(* IEC 61131-3 sources: RPA_SEM_TRYSKANI/, 5 files *)

(* ---- piskovani_new_pokus.st ---- *)
TYPE
  SuperStatesEnum : (ST_INICIALIZACE, ST_RESET_POSITION_OF_MOTORS, ST_WAIT_FOR_COMMAND, ST_MODE_SELECTION, ST_MANUAL_MODE, ST_AUTOMATIC_MODE, ST_CHECK_POSITION_OF_MOTORS, ST_STOP, ST_EMERGENCY_STOP) := ST_INICIALIZACE;
END_TYPE

PROGRAM SuperStavy
  VAR
    I_Start AT %IX0.6 : BOOL := 1;
    I_PowerOn AT %IX1.1 : BOOL := 1;
    I_StopBtn AT %IX1.2 : BOOL;
    I_StopResBtn AT %IX1.3 : BOOL;
    I_EmStopBtn AT %IX1.4 : BOOL;
    I_EmStopResBtn AT %IX1.5 : BOOL;
    I_ManualSelector AT %IX1.6 : BOOL;
    I_AutomaticSelector AT %IX1.7 : BOOL := 1;
  END_VAR
  VAR
    SuperStates : SuperStatesEnum := ST_INICIALIZACE;
  END_VAR
  VAR
    I_A0 AT %IX0.0 : BOOL;
    I_A1 AT %IX0.1 : BOOL;
    I_B0 AT %IX0.2 : BOOL;
    I_B1 AT %IX0.3 : BOOL;
    I_C0 AT %IX0.4 : BOOL;
    I_C1 AT %IX0.5 : BOOL;
  END_VAR
  VAR
    I_Qt : BOOL;
  END_VAR
  VAR
    Q_A AT %QX0.4 : BOOL;
    Q_B AT %QX0.5 : BOOL;
    Q_C AT %QX0.6 : BOOL;
  END_VAR
  VAR
    Q_PositionOk : BOOL;
    Q_PositionNotOk : BOOL;
    Q_It : BOOL;
    InputArr : ARRAY [0..7] OF BYTE;
    InputWord : INT;
    TRANS_MATX : ARRAY [0..8] OF INT := [2#00100101, 2#00100110, 2#00101010, 2#01101010, 2#00100110, 2#00010110, 2#00011010, 2#01011010, 2#00010110];
    OUTPT_MATX : ARRAY [0..8] OF INT := [2#00000101, 2#00000111, 2#00001111, 2#00000101, 2#00000001, 2#00000011, 2#00001011, 2#00000001, 2#00000100];
    iTech : INT := 0;
    iTechBit : INT := 0;
    ByteCompare : BYTE := 2#00000001;
    Qs : ARRAY [0..7] OF BOOL;
    TechnologicalSequenceState : INT := 0;
    SuperSequenceState : INT := 1;
    TON_0 : TON;
    BlastingTime : TIME := t#5s;
  END_VAR

  (*IF (I_EMSTOPBTN = true) THEN

      SuperStates := ST_EMERGENCY_STOP;

  END_IF;*)

  IF (I_Start = true) THEN

      SuperStates := ST_INICIALIZACE;

  ELSE
      SuperStates := ST_STOP;

  END_IF;

  CASE SuperStates OF

    ST_INICIALIZACE:
      (*SuperSequenceState := 1;
      IF (I_Start = true) THEN (*Uprava 06.05.2021*)

        (*SuperStates := ST_RESET_POSITION_OF_MOTORS;

      END_IF;*)

      SuperStates := ST_RESET_POSITION_OF_MOTORS;

    ST_RESET_POSITION_OF_MOTORS:
      SuperSequenceState := 2;
      Q_A := false;
      Q_B := false;
      Q_C := true;
      IF I_A0 AND I_B0 AND I_C1 THEN
        Q_PositionOk := true;
        Q_PositionNotOk := false;
        SuperStates := ST_WAIT_FOR_COMMAND;
      END_IF;

    ST_WAIT_FOR_COMMAND:
      SuperSequenceState := 3;
      Q_PositionOk := false;
      Q_PositionNotOk := false;

      SuperStates := ST_MODE_SELECTION;

    ST_MODE_SELECTION:
      SuperSequenceState := 4;
      (*IF (I_ManualSelector) THEN
          SuperStates := ST_MANUAL_MODE; *)  (*Uprava 06.05.2021*)
      (*ELSIF (I_AutomaticSelector) THEN *)
      IF (I_Start = true) THEN
          SuperStates := ST_AUTOMATIC_MODE;
      ELSIF (I_ManualSelector = true) AND (I_Start = true) THEN
          SuperStates := ST_MANUAL_MODE;
      END_IF;

      (*END_IF;*)    (*Uprava 06.05.2021*)
      (*TODO// Comeback from this state to STOP*)

    ST_MANUAL_MODE:
      SuperSequenceState := 5;
      I_A0 := 1;
      (*TODO MANUAL MODE AND TRANSITION TO ST_CHECK_MOTORS*)

    ST_AUTOMATIC_MODE:
      SuperSequenceState := 6;

      (*  Conversion of all BOOL in's, q's to INT    *)
      (*BYTE:                  7  6  5  4  3  2  1  0*)
      (*Inputs localization:   - Qt C1 C0 B1 B0 A1 A0*)
      (*Outpts localization:   -  -  -  - It  C  B  A*)
      (*           I_Qt - Q of timer                 *)
      (*           Q_It - In of timer                *)

      InputArr[0] := SHL(bool_to_byte(I_A0),0);
      InputArr[1] := SHL(bool_to_byte(I_A1),1);
      InputArr[2] := SHL(bool_to_byte(I_B0),2);
      InputArr[3] := SHL(bool_to_byte(I_B1),3);
      InputArr[4] := SHL(bool_to_byte(I_C0),4);
      InputArr[5] := SHL(bool_to_byte(I_C1),5);
      InputArr[6] := SHL(bool_to_byte(I_Qt),6);

      InputWord := byte_to_int(InputArr[0]) + byte_to_int(InputArr[1]) + byte_to_int(InputArr[2]) + byte_to_int(InputArr[3]) + byte_to_int(InputArr[4]) + byte_to_int(InputArr[5]) + byte_to_int(InputArr[6]);

      (*   End of Conversion   *)

      IF (InputWord = TRANS_MATX[iTech]) THEN

        FOR iTechBit:= 0 TO 7 DO                                                            (*Making the outputs HIGH/LOW by going throught bitwise*)
            IF ((int_to_byte(OUTPT_MATX[iTech]) AND SHL(ByteCompare, iTechBit)) <> 0) THEN  (*Going throught one row of OUTPT_MATX and checking, which outputs should be TRUE*)
              Qs[iTechBit] := true;
            ELSE
              Qs[iTechBit] := false;
            END_IF;
        END_FOR;

        (*Mapping of outputs*)
        Q_A := Qs[0];
        Q_B := Qs[1];
        Q_C := Qs[2];
        Q_It := Qs[3];
        (*End of mapping of outputs*)

        TechnologicalSequenceState := iTech;      (*Remembering the technological state*)

        iTech := iTech + 1;                       (*Going to the next state*)

      END_IF;

      (*Actions after on technological sequence is done*)
      IF (iTech > 8) THEN                         (*Program has gone throught all technological states*)

        iTech := 0;                               (*Reset sequence*)
      END_IF;

     (*ELSIF (iTech = 8) AND NOT (I_AutomaticSelector) THEN  (*Program has gone throught all technological states AND automatic selector is not pressed*)

      (*  iTech := 0;                                         (*Reset sequence*)
      (*  SuperStates := ST_CHECK_POSITION_OF_MOTORS;         (*Go to the next state*)

      (*ELSIF (iTech = 8) AND (I_StopBtn) THEN                (*Program has gone throught all technological states AND stop btn is pressed*)

       (* SuperStates := ST_STOP;                               (*Go to stop state*)

     (* END_IF;*)

    ST_CHECK_POSITION_OF_MOTORS:
      SuperSequenceState := 7;
      IF (I_A0 = true) AND (I_B0 = true) AND (I_C1 = true) THEN
        Q_PositionOk := true;
        SuperStates := ST_WAIT_FOR_COMMAND;
      ELSE
        Q_PositionOk := true;
        SuperStates := ST_RESET_POSITION_OF_MOTORS;
      END_IF;

    ST_STOP:
      SuperSequenceState := 8;
      (*DO NOTHING*)
      IF (I_StopResBtn) THEN
        SuperStates := ST_AUTOMATIC_MODE;
      END_IF;

    ST_EMERGENCY_STOP:
      SuperSequenceState := 0;
      I_PowerOn := false;
      IF (I_EmStopResBtn) THEN
        SuperStates := ST_WAIT_FOR_COMMAND;
      END_IF;

  END_CASE;

  (*Function block calling*)

  TON_0(IN := I_B1, PT := BlastingTime, Q => I_Qt);

  (*End of Function block calling*)

END_PROGRAM

CONFIGURATION Config0

  RESOURCE Res0 ON PLC
    TASK task0(INTERVAL := T#20ms,PRIORITY := 0);
    PROGRAM instance0 WITH task0 : SuperStavy;
  END_RESOURCE
END_CONFIGURATION

(* ---- SuperstavyAllBugsFix.st ---- *)
TYPE
  SuperStatesEnum : (ST_INICIALIZACE, ST_RESET_POSITION_OF_MOTORS, ST_WAIT_FOR_COMMAND, ST_MODE_SELECTION, ST_MANUAL_MODE, ST_AUTOMATIC_MODE, ST_CHECK_POSITION_OF_MOTORS, ST_STOP, ST_EMERGENCY_STOP) := ST_INICIALIZACE;
END_TYPE

PROGRAM SuperStavy
  VAR
    I_Start : BOOL := 0;
  END_VAR
  VAR
    I_StartScada AT %MW0 : INT := 0;
  END_VAR
  VAR
    I_PowerOn : BOOL := 1;
    I_StopBtn : BOOL;
  END_VAR
  VAR
    Q_StopBulbScada AT %MW7 : INT;
  END_VAR
  VAR
    I_StopResBtn : BOOL;
    I_EmStopBtn : BOOL;
  END_VAR
  VAR
    I_EmStopBtnScada AT %MW4 : INT;
  END_VAR
  VAR
    I_EmStopResBtn : BOOL;
  END_VAR
  VAR
    I_EmStopResBtnScada AT %MW2 : INT;
  END_VAR
  VAR
    I_ManualSelector : BOOL;
    I_AutomaticSelector : BOOL := 1;
    SuperStates : SuperStatesEnum;
  END_VAR
  VAR
    I_A0 AT %IX0.0 : BOOL;
    I_A1 AT %IX0.1 : BOOL;
    I_B0 AT %IX0.2 : BOOL;
    I_B1 AT %IX0.3 : BOOL;
    I_C0 AT %IX0.4 : BOOL;
    I_C1 AT %IX0.5 : BOOL;
  END_VAR
  VAR
    I_Qt : BOOL;
  END_VAR
  VAR
    Q_A AT %QX0.4 : BOOL;
    Q_B AT %QX0.5 : BOOL;
    Q_C AT %QX0.6 : BOOL;
  END_VAR
  VAR
    Q_PositionOk : BOOL;
    Q_PositionNotOk : BOOL;
    Q_It : BOOL;
    InputArr : ARRAY [0..7] OF BYTE;
  END_VAR
  VAR
    InputWord AT %MW5 : INT;
  END_VAR
  VAR
    TRANS_MATX : ARRAY [0..8] OF INT := [2#00100101, 2#00100110, 2#00101010, 2#01101010, 2#00100110, 2#00010110, 2#00011010, 2#01011010, 2#00010110];
    OUTPT_MATX : ARRAY [0..8] OF INT := [2#00000101, 2#00000111, 2#00001111, 2#00000101, 2#00000001, 2#00000011, 2#00001011, 2#00000001, 2#00000100];
  END_VAR
  VAR
    iTech AT %MW6 : INT := 0;
  END_VAR
  VAR
    iTechBit : INT := 0;
    ByteCompare : BYTE := 2#00000001;
    Qs : ARRAY [0..7] OF BOOL;
    TechnologicalSequenceState : INT := 0;
    SuperSequenceState : INT := 1;
  END_VAR
  VAR
    SuperSequenceStateScada AT %MW3 : INT := 0;
  END_VAR
  VAR
    TON_0 : TON;
    BlastingTime : TIME := t#5s;
  END_VAR

  IF (I_EMSTOPBTN = true) THEN

      SuperStates := ST_EMERGENCY_STOP;

  END_IF;

  (*Mapping of inputs from SCADA to real inputs*)  (*Uprava: 06.12.2021*)

  I_Start := int_to_bool(I_StartScada);
  I_EmStopBtn := int_to_bool(I_EmStopBtnScada);
  I_EmStopResBtn := int_to_bool(I_EmStopResBtnScada);

  SuperSequenceStateScada := SuperSequenceState;

  (*|Mapping of inputs from SCADA to real inputs|*)

  (*Trowing state to <WAIT FOR COMMAND> afrer stop if start wasn't pressed*)

  IF (I_EMSTOPBTN = false) AND (I_START = False) AND (SuperSequenceState <> 1) AND (SuperSequenceState <> 0) THEN

    SuperStates := ST_WAIT_FOR_COMMAND;

  END_IF;

  (*|Trowing state to <WAIT FOR COMMAND> afrer stop if start wasn't pressed|*)

  CASE SuperStates OF

    ST_INICIALIZACE:
      SuperSequenceState := 1;
      IF (I_Start = true) (*AND (I_PowerOn = true)*) THEN (*Uprava 06.12.2021*)

        SuperStates := ST_RESET_POSITION_OF_MOTORS;

      END_IF;

    ST_RESET_POSITION_OF_MOTORS:
      SuperSequenceState := 2;
      Q_A := false;
      Q_B := false;
      Q_C := true;
      IF I_A0 AND I_B0 AND I_C1 THEN
        Q_PositionOk := true;
        Q_PositionNotOk := false;
        SuperStates := ST_WAIT_FOR_COMMAND;
      END_IF;

    ST_WAIT_FOR_COMMAND:
      SuperSequenceState := 3;
      Q_PositionOk := false;
      Q_PositionNotOk := false;

      SuperStates := ST_MODE_SELECTION;

    ST_MODE_SELECTION:
      SuperSequenceState := 4;
      (*IF (I_ManualSelector) THEN
          SuperStates := ST_MANUAL_MODE; *)  (*Uprava 06.05.2021*)
      (*ELSIF (I_AutomaticSelector) THEN *)
          SuperStates := ST_AUTOMATIC_MODE;
      (*END_IF;*)    (*Uprava 06.05.2021*)
      (*TODO// Comeback from this state to STOP*)

    ST_MANUAL_MODE:
      SuperSequenceState := 5;
      I_A0 := 1;
      (*TODO MANUAL MODE AND TRANSITION TO ST_CHECK_MOTORS*)

    ST_AUTOMATIC_MODE:
      SuperSequenceState := 6;

      (*  Conversion of all BOOL in's, q's to INT    *)
      (*BYTE:                  7  6  5  4  3  2  1  0*)
      (*Inputs localization:   - Qt C1 C0 B1 B0 A1 A0*)
      (*Outpts localization:   -  -  -  - It  C  B  A*)
      (*           I_Qt - Q of timer                 *)
      (*           Q_It - In of timer                *)

      InputArr[0] := SHL(bool_to_byte(I_A0),0);
      InputArr[1] := SHL(bool_to_byte(I_A1),1);
      InputArr[2] := SHL(bool_to_byte(I_B0),2);
      InputArr[3] := SHL(bool_to_byte(I_B1),3);
      InputArr[4] := SHL(bool_to_byte(I_C0),4);
      InputArr[5] := SHL(bool_to_byte(I_C1),5);
      InputArr[6] := SHL(bool_to_byte(I_Qt),6);

      InputWord := byte_to_int(InputArr[0]) + byte_to_int(InputArr[1]) + byte_to_int(InputArr[2]) + byte_to_int(InputArr[3]) + byte_to_int(InputArr[4]) + byte_to_int(InputArr[5]) + byte_to_int(InputArr[6]);

      (*   End of Conversion   *)

      IF (InputWord = TRANS_MATX[iTech]) THEN

        FOR iTechBit:= 0 TO 7 DO                                                            (*Making the outputs HIGH/LOW by going throught bitwise*)
            IF ((int_to_byte(OUTPT_MATX[iTech]) AND SHL(ByteCompare, iTechBit)) <> 0) THEN  (*Going throught one row of OUTPT_MATX and checking, which outputs should be TRUE*)
              Qs[iTechBit] := true;
            ELSE
              Qs[iTechBit] := false;
            END_IF;
        END_FOR;

        (*Mapping of outputs*)
        Q_A := Qs[0];
        Q_B := Qs[1];
        Q_C := Qs[2];
        Q_It := Qs[3];
        (*End of mapping of outputs*)

        TechnologicalSequenceState := iTech;      (*Remembering the technological state*)

        iTech := iTech + 1;                       (*Going to the next state*)

      END_IF;

      (*Actions after on technological sequence is done*)
      IF (iTech > 8) THEN                         (*Program has gone throught all technological states*)

        iTech := 0;                               (*Reset sequence*)
      END_IF;

     (*ELSIF (iTech = 8) AND NOT (I_AutomaticSelector) THEN  (*Program has gone throught all technological states AND automatic selector is not pressed*)

      (*  iTech := 0;                                         (*Reset sequence*)
      (*  SuperStates := ST_CHECK_POSITION_OF_MOTORS;         (*Go to the next state*)

      (*ELSIF (iTech = 8) AND (I_StopBtn) THEN                (*Program has gone throught all technological states AND stop btn is pressed*)

       (* SuperStates := ST_STOP;                               (*Go to stop state*)

     (* END_IF;*)

    ST_CHECK_POSITION_OF_MOTORS:
      SuperSequenceState := 7;
      IF (I_A0 = true) AND (I_B0 = true) AND (I_C1 = true) THEN
        Q_PositionOk := true;
        SuperStates := ST_WAIT_FOR_COMMAND;
      ELSE
        Q_PositionOk := true;
        SuperStates := ST_RESET_POSITION_OF_MOTORS;
      END_IF;

    ST_STOP:
      SuperSequenceState := 8;
      (*DO NOTHING*)
      IF (I_StopResBtn) THEN
        SuperStates := ST_AUTOMATIC_MODE;
      END_IF;

    ST_EMERGENCY_STOP:
      SuperSequenceState := 0;
      Q_StopBulbScada := 1;
      I_PowerOn := false;
      IF (I_EmStopResBtn = TRUE) AND (I_EmStopBtn = FALSE) THEN
        Q_StopBulbScada := 0;
        SuperStates := ST_WAIT_FOR_COMMAND;
      END_IF;

  END_CASE;

  (*Function block calling*)

  TON_0(IN := I_B1, PT := BlastingTime, Q => I_Qt);

  (*End of Function block calling*)

END_PROGRAM

CONFIGURATION Config0

  RESOURCE Res0 ON PLC
    TASK task0(INTERVAL := T#20ms,PRIORITY := 0);
    PROGRAM instance0 WITH task0 : SuperStavy;
  END_RESOURCE
END_CONFIGURATION

(* ---- SuperstavyTechSeqBugFix.st ---- *)
TYPE
  SuperStatesEnum : (ST_INICIALIZACE, ST_RESET_POSITION_OF_MOTORS, ST_WAIT_FOR_COMMAND, ST_MODE_SELECTION, ST_MANUAL_MODE, ST_AUTOMATIC_MODE, ST_CHECK_POSITION_OF_MOTORS, ST_STOP, ST_EMERGENCY_STOP) := ST_INICIALIZACE;
END_TYPE

PROGRAM SuperStavy
  VAR
    I_Start AT %IX1.0 : BOOL := 1;
    I_PowerOn AT %IX1.1 : BOOL := 1;
    I_StopBtn AT %IX1.2 : BOOL;
    I_StopResBtn AT %IX1.3 : BOOL;
    I_EmStopBtn AT %IX1.4 : BOOL;
    I_EmStopResBtn AT %IX1.5 : BOOL;
    I_ManualSelector AT %IX1.6 : BOOL;
    I_AutomaticSelector AT %IX1.7 : BOOL := 1;
  END_VAR
  VAR
    SuperStates : SuperStatesEnum;
  END_VAR
  VAR
    I_A0 AT %IX0.0 : BOOL;
    I_A1 AT %IX0.1 : BOOL;
    I_B0 AT %IX0.2 : BOOL;
    I_B1 AT %IX0.3 : BOOL;
    I_C0 AT %IX0.4 : BOOL;
    I_C1 AT %IX0.5 : BOOL;
  END_VAR
  VAR
    I_Qt : BOOL;
  END_VAR
  VAR
    Q_A AT %QX0.4 : BOOL;
    Q_B AT %QX0.5 : BOOL;
    Q_C AT %QX0.6 : BOOL;
  END_VAR
  VAR
    Q_PositionOk : BOOL;
    Q_PositionNotOk : BOOL;
    Q_It : BOOL;
    InputArr : ARRAY [0..7] OF BYTE;
    InputWord : INT;
    TRANS_MATX : ARRAY [0..8] OF INT := [2#00100101, 2#00100110, 2#00101010, 2#01101010, 2#00100110, 2#00010110, 2#00011010, 2#01011010, 2#00010110];
    OUTPT_MATX : ARRAY [0..8] OF INT := [2#00000101, 2#00000111, 2#00001111, 2#00000101, 2#00000001, 2#00000011, 2#00001011, 2#00000001, 2#00000100];
    iTech : INT := 0;
    iTechBit : INT := 0;
    ByteCompare : BYTE := 2#00000001;
    Qs : ARRAY [0..7] OF BOOL;
    TechnologicalSequenceState : INT := 0;
    SuperSequenceState : INT := 1;
    TON_0 : TON;
    BlastingTime : TIME := t#5s;
  END_VAR

  IF (I_EMSTOPBTN = true) THEN

      SuperStates := ST_EMERGENCY_STOP;

  END_IF;

  CASE SuperStates OF

    ST_INICIALIZACE:
      SuperSequenceState := 1;
      (*IF (I_Start = true) AND (I_PowerOn = true) THEN*) (*Uprava 06.05.2021*)

        SuperStates := ST_RESET_POSITION_OF_MOTORS;

      (*END_IF;*)

    ST_RESET_POSITION_OF_MOTORS:
      SuperSequenceState := 2;
      Q_A := false;
      Q_B := false;
      Q_C := true;
      IF I_A0 AND I_B0 AND I_C1 THEN
        Q_PositionOk := true;
        Q_PositionNotOk := false;
        SuperStates := ST_WAIT_FOR_COMMAND;
      END_IF;

    ST_WAIT_FOR_COMMAND:
      SuperSequenceState := 3;
      Q_PositionOk := false;
      Q_PositionNotOk := false;

      SuperStates := ST_MODE_SELECTION;

    ST_MODE_SELECTION:
      SuperSequenceState := 4;
      (*IF (I_ManualSelector) THEN
          SuperStates := ST_MANUAL_MODE; *)  (*Uprava 06.05.2021*)
      (*ELSIF (I_AutomaticSelector) THEN *)
          SuperStates := ST_AUTOMATIC_MODE;
      (*END_IF;*)    (*Uprava 06.05.2021*)
      (*TODO// Comeback from this state to STOP*)

    ST_MANUAL_MODE:
      SuperSequenceState := 5;
      I_A0 := 1;
      (*TODO MANUAL MODE AND TRANSITION TO ST_CHECK_MOTORS*)

    ST_AUTOMATIC_MODE:
      SuperSequenceState := 6;

      (*  Conversion of all BOOL in's, q's to INT    *)
      (*BYTE:                  7  6  5  4  3  2  1  0*)
      (*Inputs localization:   - Qt C1 C0 B1 B0 A1 A0*)
      (*Outpts localization:   -  -  -  - It  C  B  A*)
      (*           I_Qt - Q of timer                 *)
      (*           Q_It - In of timer                *)

      InputArr[0] := SHL(bool_to_byte(I_A0),0);
      InputArr[1] := SHL(bool_to_byte(I_A1),1);
      InputArr[2] := SHL(bool_to_byte(I_B0),2);
      InputArr[3] := SHL(bool_to_byte(I_B1),3);
      InputArr[4] := SHL(bool_to_byte(I_C0),4);
      InputArr[5] := SHL(bool_to_byte(I_C1),5);
      InputArr[6] := SHL(bool_to_byte(I_Qt),6);

      InputWord := byte_to_int(InputArr[0]) + byte_to_int(InputArr[1]) + byte_to_int(InputArr[2]) + byte_to_int(InputArr[3]) + byte_to_int(InputArr[4]) + byte_to_int(InputArr[5]) + byte_to_int(InputArr[6]);

      (*   End of Conversion   *)

      IF (InputWord = TRANS_MATX[iTech]) THEN

        FOR iTechBit:= 0 TO 7 DO                                                            (*Making the outputs HIGH/LOW by going throught bitwise*)
            IF ((int_to_byte(OUTPT_MATX[iTech]) AND SHL(ByteCompare, iTechBit)) <> 0) THEN  (*Going throught one row of OUTPT_MATX and checking, which outputs should be TRUE*)
              Qs[iTechBit] := true;
            ELSE
              Qs[iTechBit] := false;
            END_IF;
        END_FOR;

        (*Mapping of outputs*)
        Q_A := Qs[0];
        Q_B := Qs[1];
        Q_C := Qs[2];
        Q_It := Qs[3];
        (*End of mapping of outputs*)

        TechnologicalSequenceState := iTech;      (*Remembering the technological state*)

        iTech := iTech + 1;                       (*Going to the next state*)

      END_IF;

      (*Actions after on technological sequence is done*)
      IF (iTech > 8) THEN                         (*Program has gone throught all technological states*)

        iTech := 0;                               (*Reset sequence*)
      END_IF;

     (*ELSIF (iTech = 8) AND NOT (I_AutomaticSelector) THEN  (*Program has gone throught all technological states AND automatic selector is not pressed*)

      (*  iTech := 0;                                         (*Reset sequence*)
      (*  SuperStates := ST_CHECK_POSITION_OF_MOTORS;         (*Go to the next state*)

      (*ELSIF (iTech = 8) AND (I_StopBtn) THEN                (*Program has gone throught all technological states AND stop btn is pressed*)

       (* SuperStates := ST_STOP;                               (*Go to stop state*)

     (* END_IF;*)

    ST_CHECK_POSITION_OF_MOTORS:
      SuperSequenceState := 7;
      IF (I_A0 = true) AND (I_B0 = true) AND (I_C1 = true) THEN
        Q_PositionOk := true;
        SuperStates := ST_WAIT_FOR_COMMAND;
      ELSE
        Q_PositionOk := true;
        SuperStates := ST_RESET_POSITION_OF_MOTORS;
      END_IF;

    ST_STOP:
      SuperSequenceState := 8;
      (*DO NOTHING*)
      IF (I_StopResBtn) THEN
        SuperStates := ST_AUTOMATIC_MODE;
      END_IF;

    ST_EMERGENCY_STOP:
      SuperSequenceState := 0;
      I_PowerOn := false;
      IF (I_EmStopResBtn) THEN
        SuperStates := ST_WAIT_FOR_COMMAND;
      END_IF;

  END_CASE;

  (*Function block calling*)

  TON_0(IN := I_B1, PT := BlastingTime, Q => I_Qt);

  (*End of Function block calling*)

END_PROGRAM

CONFIGURATION Config0

  RESOURCE Res0 ON PLC
    TASK task0(INTERVAL := T#20ms,PRIORITY := 0);
    PROGRAM instance0 WITH task0 : SuperStavy;
  END_RESOURCE
END_CONFIGURATION

(* ---- SuperstavyTechSeqBugFixWithStart.st ---- *)
TYPE
  SuperStatesEnum : (ST_INICIALIZACE, ST_RESET_POSITION_OF_MOTORS, ST_WAIT_FOR_COMMAND, ST_MODE_SELECTION, ST_MANUAL_MODE, ST_AUTOMATIC_MODE, ST_CHECK_POSITION_OF_MOTORS, ST_STOP, ST_EMERGENCY_STOP) := ST_INICIALIZACE;
END_TYPE

PROGRAM SuperStavy
  VAR
    I_Start AT %IX0.6 : BOOL := 0;
    Start_RTRIG AT %IX0.7 : BOOL := 1;
    I_PowerOn AT %IX1.1 : BOOL := 1;
    I_StopBtn AT %IX1.2 : BOOL;
    I_StopResBtn AT %IX1.3 : BOOL;
    I_EmStopBtn AT %IX1.4 : BOOL;
    I_EmStopResBtn AT %IX1.5 : BOOL;
    I_ManualSelector AT %IX1.6 : BOOL;
    I_AutomaticSelector AT %IX1.7 : BOOL := 1;
  END_VAR
  VAR
    SuperStates : SuperStatesEnum := ST_INICIALIZACE;
  END_VAR
  VAR
    I_A0 AT %IX0.0 : BOOL;
    I_A1 AT %IX0.1 : BOOL;
    I_B0 AT %IX0.2 : BOOL;
    I_B1 AT %IX0.3 : BOOL;
    I_C0 AT %IX0.4 : BOOL;
    I_C1 AT %IX0.5 : BOOL;
  END_VAR
  VAR
    I_Qt : BOOL;
  END_VAR
  VAR
    Q_A AT %QX0.4 : BOOL;
    Q_B AT %QX0.5 : BOOL;
    Q_C AT %QX0.6 : BOOL;
  END_VAR
  VAR
    Q_PositionOk : BOOL;
    Q_PositionNotOk : BOOL;
    Q_It : BOOL;
    InputArr : ARRAY [0..7] OF BYTE;
    InputWord : INT;
  END_VAR
  VAR
    ScadaStart AT %MW0 : INT;
  END_VAR
  VAR
    TRANS_MATX : ARRAY [0..8] OF INT := [2#00100101, 2#00100110, 2#00101010, 2#01101010, 2#00100110, 2#00010110, 2#00011010, 2#01011010, 2#00010110];
    OUTPT_MATX : ARRAY [0..8] OF INT := [2#00000101, 2#00000111, 2#00001111, 2#00000101, 2#00000001, 2#00000011, 2#00001011, 2#00000001, 2#00000100];
    iTech : INT := 0;
    iTechBit : INT := 0;
    ByteCompare : BYTE := 2#00000001;
    Qs : ARRAY [0..7] OF BOOL;
    TechnologicalSequenceState : INT := 0;
    SuperSequenceState : INT;
    TON_0 : TON;
    BlastingTime : TIME := t#5s;
  END_VAR

  IF (I_EMSTOPBTN = true) THEN

        SuperStates := ST_EMERGENCY_STOP;

    END_IF;

  (*

  TODO: Write of input word from scada to logical inputs (like I_Start)

  *)

  I_Start := int_to_bool(ScadaStart);

    CASE SuperStates OF

      ST_INICIALIZACE:
        SuperSequenceState := 1;
        IF (I_Start = true) (*AND (I_PowerOn = true)*) THEN (*Uprava 10.11.2021*)

          SuperStates := ST_RESET_POSITION_OF_MOTORS;

        END_IF;

      ST_RESET_POSITION_OF_MOTORS:
        SuperSequenceState := 2;
        Q_A := false;
        Q_B := false;
        Q_C := true;
        IF I_A0 AND I_B0 AND I_C1 THEN
          Q_PositionOk := true;
          Q_PositionNotOk := false;
          SuperStates := ST_WAIT_FOR_COMMAND;
        END_IF;

      ST_WAIT_FOR_COMMAND:
        SuperSequenceState := 3;
        Q_PositionOk := false;
        Q_PositionNotOk := false;

        SuperStates := ST_MODE_SELECTION;

      ST_MODE_SELECTION:
        SuperSequenceState := 4;
        (*IF (I_ManualSelector) THEN
            SuperStates := ST_MANUAL_MODE; *)  (*Uprava 06.05.2021*)
        (*ELSIF (I_AutomaticSelector) THEN *)
            SuperStates := ST_AUTOMATIC_MODE;
        (*END_IF;*)    (*Uprava 06.05.2021*)
        (*TODO// Comeback from this state to STOP*)

      ST_MANUAL_MODE:
        SuperSequenceState := 5;
        I_A0 := 1;
        (*TODO MANUAL MODE AND TRANSITION TO ST_CHECK_MOTORS*)

      ST_AUTOMATIC_MODE:
        SuperSequenceState := 6;

        (*  Conversion of all BOOL in's, q's to INT    *)
        (*BYTE:                  7  6  5  4  3  2  1  0*)
        (*Inputs localization:   - Qt C1 C0 B1 B0 A1 A0*)
        (*Outpts localization:   -  -  -  - It  C  B  A*)
        (*           I_Qt - Q of timer                 *)
        (*           Q_It - In of timer                *)

        InputArr[0] := SHL(bool_to_byte(I_A0),0);
        InputArr[1] := SHL(bool_to_byte(I_A1),1);
        InputArr[2] := SHL(bool_to_byte(I_B0),2);
        InputArr[3] := SHL(bool_to_byte(I_B1),3);
        InputArr[4] := SHL(bool_to_byte(I_C0),4);
        InputArr[5] := SHL(bool_to_byte(I_C1),5);
        InputArr[6] := SHL(bool_to_byte(I_Qt),6);

        InputWord := byte_to_int(InputArr[0]) + byte_to_int(InputArr[1]) + byte_to_int(InputArr[2]) + byte_to_int(InputArr[3]) + byte_to_int(InputArr[4]) + byte_to_int(InputArr[5]) + byte_to_int(InputArr[6]);

        (*   End of Conversion   *)

        IF (InputWord = TRANS_MATX[iTech]) THEN

          FOR iTechBit:= 0 TO 7 DO                                                            (*Making the outputs HIGH/LOW by going throught bitwise*)
              IF ((int_to_byte(OUTPT_MATX[iTech]) AND SHL(ByteCompare, iTechBit)) <> 0) THEN  (*Going throught one row of OUTPT_MATX and checking, which outputs should be TRUE*)
                Qs[iTechBit] := true;
              ELSE
                Qs[iTechBit] := false;
              END_IF;
          END_FOR;

          (*Mapping of outputs*)
          Q_A := Qs[0];
          Q_B := Qs[1];
          Q_C := Qs[2];
          Q_It := Qs[3];
          (*End of mapping of outputs*)

          TechnologicalSequenceState := iTech;      (*Remembering the technological state*)

          iTech := iTech + 1;                       (*Going to the next state*)

        END_IF;

        (*Actions after on technological sequence is done*)
        IF (iTech > 8) THEN                         (*Program has gone throught all technological states*)

          iTech := 0;                               (*Reset sequence*)
        END_IF;

       (*ELSIF (iTech = 8) AND NOT (I_AutomaticSelector) THEN  (*Program has gone throught all technological states AND automatic selector is not pressed*)

        (*  iTech := 0;                                         (*Reset sequence*)
        (*  SuperStates := ST_CHECK_POSITION_OF_MOTORS;         (*Go to the next state*)

        (*ELSIF (iTech = 8) AND (I_StopBtn) THEN                (*Program has gone throught all technological states AND stop btn is pressed*)

         (* SuperStates := ST_STOP;                               (*Go to stop state*)

       (* END_IF;*)

      ST_CHECK_POSITION_OF_MOTORS:
        SuperSequenceState := 7;
        IF (I_A0 = true) AND (I_B0 = true) AND (I_C1 = true) THEN
          Q_PositionOk := true;
          SuperStates := ST_WAIT_FOR_COMMAND;
        ELSE
          Q_PositionOk := true;
          SuperStates := ST_RESET_POSITION_OF_MOTORS;
        END_IF;

      ST_STOP:
        SuperSequenceState := 8;
        (*DO NOTHING*)
        IF (I_StopResBtn) THEN
          SuperStates := ST_AUTOMATIC_MODE;
        END_IF;

      ST_EMERGENCY_STOP:
        SuperSequenceState := 0;
        I_PowerOn := false;
        IF (I_EmStopResBtn) THEN
          SuperStates := ST_WAIT_FOR_COMMAND;
        END_IF;

    END_CASE;

    (*Function block calling*)

    TON_0(IN := I_B1, PT := BlastingTime, Q => I_Qt);

    (*End of Function block calling*)
END_PROGRAM

CONFIGURATION Config0

  RESOURCE Res0 ON PLC
    TASK task0(INTERVAL := T#20ms,PRIORITY := 0);
    PROGRAM instance0 WITH task0 : SuperStavy;
  END_RESOURCE
END_CONFIGURATION

(* ---- TechSeqSemDigDvojce.st ---- *)
TYPE
  SuperStatesEnum : (ST_INICIALIZACE, ST_RESET_POSITION_OF_MOTORS, ST_WAIT_FOR_COMMAND, ST_MODE_SELECTION, ST_MANUAL_MODE, ST_AUTOMATIC_MODE, ST_CHECK_POSITION_OF_MOTORS, ST_STOP, ST_EMERGENCY_STOP) := ST_INICIALIZACE;
END_TYPE

PROGRAM SuperStavy
  VAR
    I_Start AT %IX0.5 : BOOL;
  END_VAR
  VAR
    I_PowerOn : BOOL;
    I_StopBtn : BOOL;
    I_StopResBtn : BOOL;
    I_EmStopBtn : BOOL;
    I_EmStopResBtn : BOOL;
    I_ManualSelector : BOOL;
    I_AutomaticSelector : BOOL;
    SuperStates : SuperStatesEnum;
  END_VAR
  VAR
    I_A0 AT %IX0.0 : BOOL;
    I_A1 AT %IX0.1 : BOOL;
    I_B0 AT %IX0.2 : BOOL;
    I_B1 AT %IX0.3 : BOOL;
    I_C0 AT %IX0.4 : BOOL;
  END_VAR
  VAR
    I_C1 : BOOL;
    I_Qt : BOOL;
  END_VAR
  VAR
    Q_A AT %QX0.0 : BOOL;
    Q_B AT %QX0.1 : BOOL;
    Q_C AT %QX0.2 : BOOL;
  END_VAR
  VAR
    Q_PositionOk : BOOL;
    Q_PositionNotOk : BOOL;
    Q_It : BOOL;
    InputArr : ARRAY [0..7] OF BYTE;
    InputWord : INT;
    TRANS_MATX : ARRAY [0..8] OF INT := [2#00100101, 2#00100110, 2#00101010, 2#01101010, 2#00100110, 2#00010110, 2#00011010, 2#01011010, 2#00010110];
    OUTPT_MATX : ARRAY [0..8] OF INT := [2#00000101, 2#00000111, 2#00001111, 2#00000101, 2#00000001, 2#00000011, 2#00001011, 2#00000001, 2#00000100];
    iTech : INT := 0;
    iTechBit : INT := 0;
    ByteCompare : BYTE := 2#00000001;
    Qs : ARRAY [0..7] OF BOOL;
    TechnologicalSequenceState : INT := 0;
    SuperSequenceState : INT := 1;
    TON_0 : TON;
    BlastingTime : TIME := t#5s;
  END_VAR

  IF (I_EMSTOPBTN = true) THEN

      SuperStates := ST_EMERGENCY_STOP;

  END_IF;

  CASE SuperStates OF

    ST_INICIALIZACE:
      SuperSequenceState := 1;
      IF (I_Start = true)(* AND (I_PowerOn = true)*) THEN (*Uprava: 07.05.21*)

        SuperStates := ST_RESET_POSITION_OF_MOTORS;

      END_IF;

    ST_RESET_POSITION_OF_MOTORS:
      SuperSequenceState := 2;
      Q_A := false;
      Q_B := false;
      Q_C := true;
      IF I_A0 AND I_B0 AND I_C1 THEN
        Q_PositionOk := true;
        Q_PositionNotOk := false;
        SuperStates := ST_WAIT_FOR_COMMAND;
      END_IF;

    ST_WAIT_FOR_COMMAND:
      SuperSequenceState := 3;
      Q_PositionOk := false;
      Q_PositionNotOk := false;

      SuperStates := ST_MODE_SELECTION;

    ST_MODE_SELECTION:
      (*SuperSequenceState := 4;
      IF (I_ManualSelector) THEN
          SuperStates := ST_MANUAL_MODE;
      ELSIF (I_AutomaticSelector) THEN*)
          SuperStates := ST_AUTOMATIC_MODE;
      (*END_IF;*)   (*Uprava: 07.05.21*)
      (*TODO// Comeback from this state to STOP*)

    ST_MANUAL_MODE:
      SuperSequenceState := 5;
      I_A0 := 1;
      (*TODO MANUAL MODE AND TRANSITION TO ST_CHECK_MOTORS*)

    ST_AUTOMATIC_MODE:
      SuperSequenceState := 6;

      (*  Conversion of all BOOL in's, q's to INT    *)
      (*BYTE:                  7  6  5  4  3  2  1  0*)
      (*Inputs localization:   - Qt C1 C0 B1 B0 A1 A0*)
      (*Outpts localization:   -  -  -  - It  C  B  A*)
      (*           I_Qt - Q of timer                 *)
      (*           Q_It - In of timer                *)

      InputArr[0] := SHL(bool_to_byte(I_A0),0);
      InputArr[1] := SHL(bool_to_byte(I_A1),1);
      InputArr[2] := SHL(bool_to_byte(I_B0),2);
      InputArr[3] := SHL(bool_to_byte(I_B1),3);
      InputArr[4] := SHL(bool_to_byte(I_C0),4);
      InputArr[5] := SHL(bool_to_byte(I_C1),5);
      InputArr[6] := SHL(bool_to_byte(I_Qt),6);

      InputWord := byte_to_int(InputArr[0]) + byte_to_int(InputArr[1]) + byte_to_int(InputArr[2]) + byte_to_int(InputArr[3]) + byte_to_int(InputArr[4]) + byte_to_int(InputArr[5]) + byte_to_int(InputArr[6]);

      (*   End of Conversion   *)

      IF (InputWord = TRANS_MATX[iTech]) THEN

        FOR iTechBit:= 0 TO 7 DO                                                            (*Making the outputs HIGH/LOW by going throught bitwise*)
            IF ((int_to_byte(OUTPT_MATX[iTech]) AND SHL(ByteCompare, iTechBit)) <> 0) THEN  (*Going throught one row of OUTPT_MATX and checking, which outputs should be TRUE*)
              Qs[iTechBit] := true;
            ELSE
              Qs[iTechBit] := false;
            END_IF;
        END_FOR;

        (*Mapping of outputs*)
        Q_A := Qs[0];
        Q_B := Qs[1];
        Q_C := Qs[2];
        Q_It := Qs[3];
        (*End of mapping of outputs*)

        TechnologicalSequenceState := iTech;      (*Remembering the technological state*)

        iTech := iTech + 1;                       (*Going to the next state*)

      END_IF;

      (*Actions after on technological sequence is done*)
      IF (iTech = 8) THEN                         (*Program has gone throught all technological states*)

        iTech := 0;                               (*Reset sequence*)

      (*ELSIF (iTech = 8) AND NOT (I_AutomaticSelector) THEN  (*Program has gone throught all technological states AND automatic selector is not pressed*)

       (* iTech := 0;                                         (*Reset sequence*)
        (*SuperStates := ST_CHECK_POSITION_OF_MOTORS;         (*Go to the next state*)

      (*ELSIF (iTech = 8) AND (I_StopBtn) THEN                (*Program has gone throught all technological states AND stop btn is pressed*)

        (*SuperStates := ST_STOP;                             (*Go to stop state*)
        (*Uprava: 07.05.21*)

      END_IF;

    ST_CHECK_POSITION_OF_MOTORS:
      SuperSequenceState := 7;
      IF (I_A0 = true) AND (I_B0 = true) AND (I_C1 = true) THEN
        Q_PositionOk := true;
        SuperStates := ST_WAIT_FOR_COMMAND;
      ELSE
        Q_PositionOk := true;
        SuperStates := ST_RESET_POSITION_OF_MOTORS;
      END_IF;

    ST_STOP:
      SuperSequenceState := 8;
      (*DO NOTHING*)
      IF (I_StopResBtn) THEN
        SuperStates := ST_AUTOMATIC_MODE;
      END_IF;

    ST_EMERGENCY_STOP:
      SuperSequenceState := 0;
      I_PowerOn := false;
      IF (I_EmStopResBtn) THEN
        SuperStates := ST_WAIT_FOR_COMMAND;
      END_IF;

  END_CASE;

  (*Function block calling*)

  TON_0(IN := I_B1, PT := BlastingTime, Q => I_Qt);

  (*End of Function block calling*)

END_PROGRAM

CONFIGURATION Config0

  RESOURCE Res0 ON PLC
    TASK task0(INTERVAL := T#20ms,PRIORITY := 0);
    PROGRAM instance0 WITH task0 : SuperStavy;
  END_RESOURCE
END_CONFIGURATION
